FUNCTION_BLOCK AE_TO_AE_AX_SPLIT (* Relays a unidirectional AE Socket onward as a bidirectional AE_AX Plug (Trigger passthrough), plus an extra AX Plug mirroring the AE_AX backward (state) channel *)
  (* Standard: 61499-2; Function: Any Event coming in by IN is forwarded to OUT unchanged; the backward Event/Bool fired into OUT by the downstream Socket is mirrored out via AX_OUT (IN has no backward channel to relay it back to); Description: Copyright (c) 2026 HR Agrartechnik GmbH This program and the accompanying materials are made available under the terms of the Eclipse Public License 2.0 which is available at https://www.eclipse.org/legal/epl-2.0/ SPDX-License-Identifier: EPL-2.0 *)
  (* Version 1.0, 2026-09-04, Franz Höpfinger, HR Agrartechnik GmbH, Initial Version *)
  PACKAGE adapter::events::bidirectional;
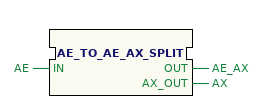
  SOCKETS
    IN : adapter::types::unidirectional::AE; (* Input (Trigger, unidirectional) *)
  END_SOCKETS
  PLUGS
    OUT : adapter::types::bidirectional::AE_AX; (* Output (Trigger out, Zustand in) *)
    AX_OUT : adapter::types::unidirectional::AX; (* mirrors the AE_AX backward (state) channel *)
  END_PLUGS
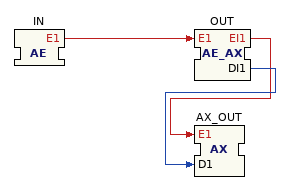
  EVENT_CONNECTIONS
    IN.E1 TO OUT.E1;
    OUT.EI1 TO AX_OUT.E1;
  END_CONNECTIONS
  DATA_CONNECTIONS
    OUT.DI1 TO AX_OUT.D1;
  END_CONNECTIONS
END_FUNCTION_BLOCK
